FUNCTION_BLOCK GR_CMD
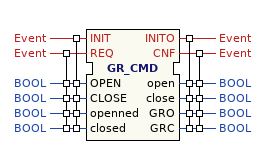
  EVENT_INPUT
    INIT WITH OPEN, CLOSE, openned, closed;
    REQ WITH OPEN, CLOSE, openned, closed;
  END_EVENT
  EVENT_OUTPUT
    INITO WITH open, close, GRO, GRC;
    CNF WITH open, close, GRO, GRC;
  END_EVENT
  VAR_INPUT
    OPEN : BOOL;
    CLOSE : BOOL;
    openned : BOOL;
    closed : BOOL;
  END_VAR
  VAR_OUTPUT
    open : BOOL;
    close : BOOL;
    GRO : BOOL;
    GRC : BOOL;
  END_VAR
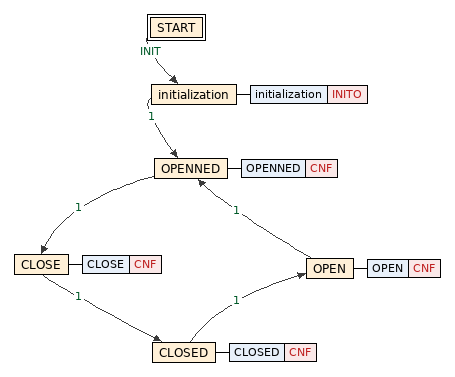
  EC_STATES
    START;
    initialization : initialization -> INITO;
    OPEN : OPEN -> CNF;
    CLOSE : CLOSE -> CNF;
    OPENNED : OPENNED -> CNF;
    CLOSED : CLOSED -> CNF;
  END_STATES
  EC_TRANSITIONS
    initialization TO OPENNED := 1;
    OPEN TO OPENNED := 1;
    CLOSE TO CLOSED := 1;
    OPENNED TO CLOSE := 1;
    CLOSED TO OPEN := 1;
    START TO initialization := INIT;
  END_TRANSITIONS
  ALGORITHM initialization IN ST:
open := TRUE;&#38;#10;close := FALSE;&#38;#10;
  END_ALGORITHM
  ALGORITHM OPEN IN ST:
open := TRUE;&#38;#10;close := FALSE;&#38;#10;
  END_ALGORITHM
  ALGORITHM CLOSE IN ST:
open := FALSE;&#38;#10;close := TRUE;&#38;#10;
  END_ALGORITHM
  ALGORITHM OPENNED IN ST:
GRO := TRUE;&#38;#10;GRC := FALSE;&#38;#10;
  END_ALGORITHM
  ALGORITHM CLOSED IN ST:
GRO := FALSE;&#38;#10;GRC := TRUE;&#38;#10;
  END_ALGORITHM
END_FUNCTION_BLOCK
